(* IEC 61131-3 sources: CodesysTest/alpha/export/FBs/Motors/Applied Motion/FB_AppliedMotionStepServoEIPPassthrough.pou, 1 file *)

(* ---- AllowClamping.m.st ---- *)
(*#-#-#-#-#-#-#-#-#-#---Declaration---#-#-#-#-#-#-#-#-#-#-#-#-#*)

METHOD AllowClamping
VAR_INPUT
END_VAR
(*#-#-#-#-#-#-#-#-#-#---Implementation---#-#-#-#-#-#-#-#-#-#-#-#-#*)

sclCommand := 16#434D; // CM Control Mode
parameter1 := 1;

commandSuccessful := FALSE;
commands.SendHostCommand := TRUE;
